// TIA Portal V18 program export: 2 tag tables, 0 data types, 2 data blocks, 3 code blocks (in call order from the OBs), 0 instance data blocks

VAR_GLOBAL   // PLC tag table "Default tag table"
   AD AT %MD6 : Real;
END_VAR

VAR_GLOBAL   // PLC tag table "PLC1_Tags"
   Start_Cmd AT %M0.0 : Bool;
   Stop_Cmd AT %M0.1 : Bool;
   bMotorRunning AT %M0.2 : Bool;
   Reset_Cmd AT %M0.3 : Bool;
   DIR_Cmd AT %M0.4 : Bool;
   PID_Setpoint AT %MD10 : Real;
   PID_ProcessValue AT %MD14 : Real;
   PID_Output AT %MD18 : Real;
   Speed_SP_toSend AT %MD22 : Real;
   Speed_PV_from2 AT %MD26 : Real;
   ATV12_Status AT %MW30 : Word;
   Control_Byte AT %MB32 : Byte;
   Clock_1Hz AT %M100.5 : Bool;
   GET_NDR AT %M1.0 : Bool;
   GET_Error AT %M1.1 : Bool;
   GET_Status AT %MW2 : Word;
   PUT_NDR AT %M1.2 : Bool;
   PUT_Error AT %M1.3 : Bool;
   PUT_Status AT %MW4 : Word;
END_VAR

DATA_BLOCK "DB10_NhanTuPLC2"   // DB10
{ S7_Optimized_Access := 'FALSE' }
VERSION : 0.1
// stored: AutoNumber true, IsOnlyStoredInLoadMemory false, IsWriteProtectedInAS false
   VAR
      Speed_Actual_fromPLC2 : Real;
      ATV12_Status_fromPLC2 : Word;
   END_VAR
BEGIN
END_DATA_BLOCK

DATA_BLOCK "DB11_GuiSangPLC2"   // DB11
{ S7_Optimized_Access := 'FALSE' }
VERSION : 0.1
// stored: AutoNumber true, IsOnlyStoredInLoadMemory false, IsWriteProtectedInAS false
   VAR
      Speed_SP_toSend : Real;
      Control_Byte_toSend : Bool;
      Reset_Cmd_toSend : Bool;
      DIR_Cmd_toSend : Bool;
   END_VAR
BEGIN
END_DATA_BLOCK

ORGANIZATION_BLOCK "Main"   // OB1, LAD, ProgramCycle
TITLE = "Main Program Sweep (Cycle)"
{ S7_Optimized_Access := 'TRUE' }
VERSION : 0.1
// stored: AutoNumber true, IsIECCheckEnabled false, SetENOAutomatically false
   VAR_INPUT
      Initial_Call : Bool;   // Initial call of this OB
      Remanence : Bool;   // =True, if remanent data are available
   END_VAR
BEGIN

REGION Network 1: Call FC_PLC1_Logic
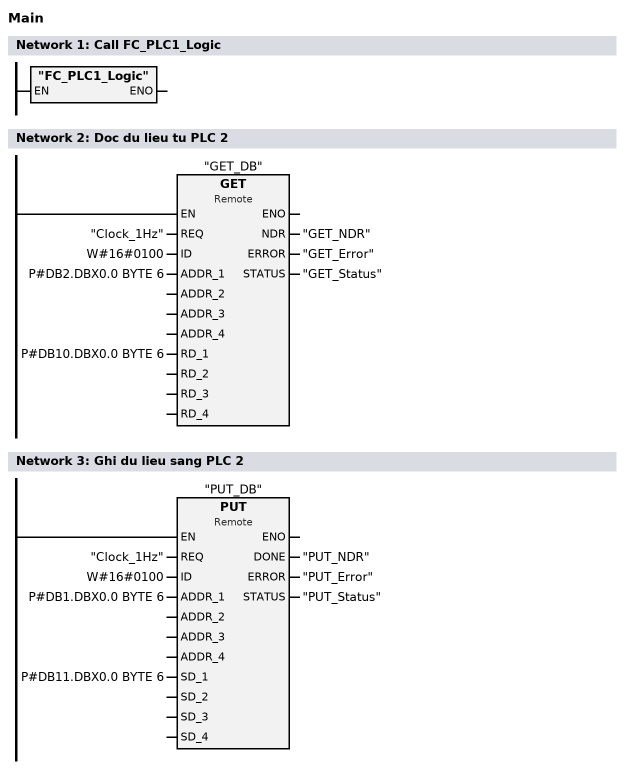
   RUNG wire#powerrail
      "FC_PLC1_Logic"()
   END_RUNG
   // the same network as SCL:
   "FC_PLC1_Logic"();
END_REGION

REGION Network 2: Doc du lieu tu PLC 2
   RUNG wire#powerrail
      { S7_Templates := "[remote_type := Remote, local_type := Variant]" } "GET_DB".GET(REQ := "Clock_1Hz", ID := W#16#0100, ADDR_1 := P#DB2.DBX0.0 BYTE 6, ADDR_2 :=, ADDR_3 :=, ADDR_4 :=, RD_1 := P#DB10.DBX0.0 BYTE 6, RD_2 :=, RD_3 :=, RD_4 :=, NDR => "GET_NDR", ERROR => "GET_Error", STATUS => "GET_Status")
   END_RUNG
   // the same network as SCL:
   "GET_DB"(REQ := "Clock_1Hz",   // GET
            ID := W#16#0100,
            ADDR_1 := P#DB2.DBX0.0 BYTE 6,
            RD_1 := P#DB10.DBX0.0 BYTE 6,
            NDR => "GET_NDR",
            ERROR => "GET_Error",
            STATUS => "GET_Status");
END_REGION

REGION Network 3: Ghi du lieu sang PLC 2
   RUNG wire#powerrail
      { S7_Templates := "[remote_type := Remote, local_type := Variant]" } "PUT_DB".PUT(REQ := "Clock_1Hz", ID := W#16#0100, ADDR_1 := P#DB1.DBX0.0 BYTE 6, ADDR_2 :=, ADDR_3 :=, ADDR_4 :=, SD_1 := P#DB11.DBX0.0 BYTE 6, SD_2 :=, SD_3 :=, SD_4 :=, DONE => "PUT_NDR", ERROR => "PUT_Error", STATUS => "PUT_Status")
   END_RUNG
   // the same network as SCL:
   "PUT_DB"(REQ := "Clock_1Hz",   // PUT
            ID := W#16#0100,
            ADDR_1 := P#DB1.DBX0.0 BYTE 6,
            SD_1 := P#DB11.DBX0.0 BYTE 6,
            DONE => "PUT_NDR",
            ERROR => "PUT_Error",
            STATUS => "PUT_Status");
END_REGION
END_ORGANIZATION_BLOCK

FUNCTION "FC_PLC1_Logic" : Void   // FC10, LAD
{ S7_Optimized_Access := 'TRUE' }
VERSION : 0.1
// stored: AutoNumber true, IsIECCheckEnabled false, SetENOAutomatically false, UDAEnableTagReadback false
BEGIN

REGION Network 1: Start Motor - Set bMotorRunning
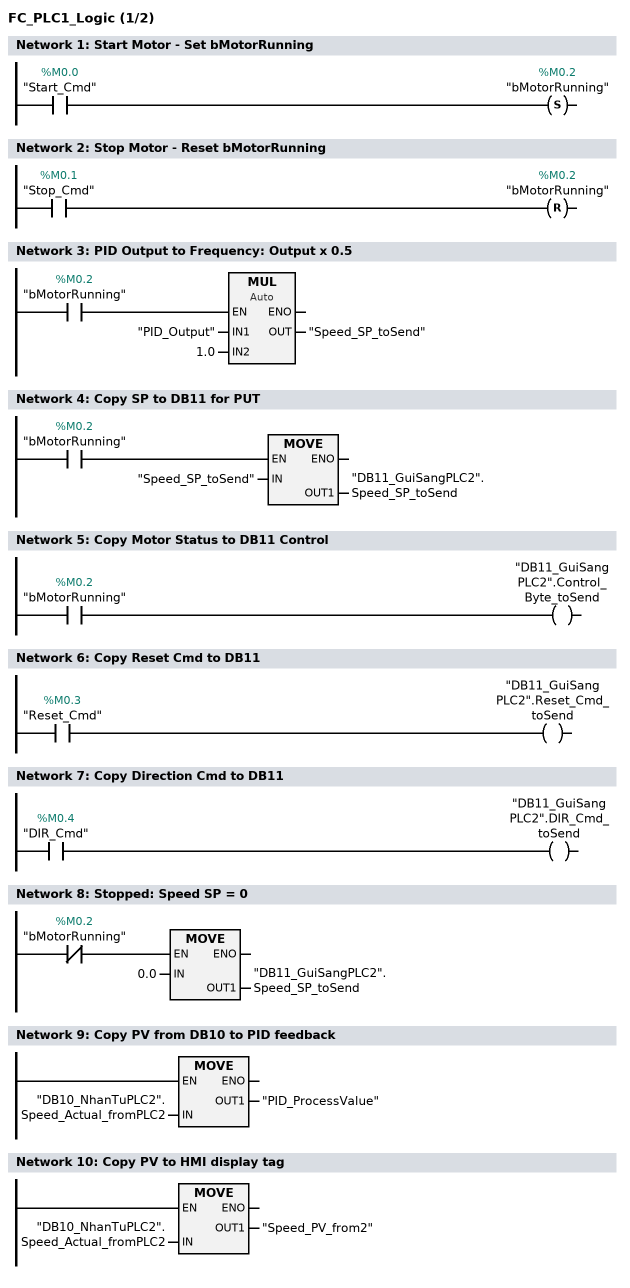
   RUNG wire#powerrail
      Contact( "Start_Cmd" )
      S_Coil( "bMotorRunning" )
   END_RUNG
   // the same network as SCL:
   IF "Start_Cmd" THEN "bMotorRunning" := TRUE; END_IF;
END_REGION

REGION Network 2: Stop Motor - Reset bMotorRunning
   RUNG wire#powerrail
      Contact( "Stop_Cmd" )
      R_Coil( "bMotorRunning" )
   END_RUNG
   // the same network as SCL:
   IF "Stop_Cmd" THEN "bMotorRunning" := FALSE; END_IF;
END_REGION

REGION Network 3: PID Output to Frequency: Output x 0.5
   RUNG wire#powerrail
      Contact( "bMotorRunning" )
      { S7_GenerateENO := "TRUE" } Mul(in1 := "PID_Output", in2 := 1.0, out => "Speed_SP_toSend")
   END_RUNG
   // the same network as SCL:
   IF "bMotorRunning" THEN "Speed_SP_toSend" := "PID_Output" * 1.0; END_IF;
END_REGION

REGION Network 4: Copy SP to DB11 for PUT
   RUNG wire#powerrail
      Contact( "bMotorRunning" )
      { S7_GenerateENO := "TRUE" } Move(in := "Speed_SP_toSend", out1 => "DB11_GuiSangPLC2".Speed_SP_toSend)
   END_RUNG
   // the same network as SCL:
   IF "bMotorRunning" THEN "DB11_GuiSangPLC2".Speed_SP_toSend := "Speed_SP_toSend"; END_IF;
END_REGION

REGION Network 5: Copy Motor Status to DB11 Control
   RUNG wire#powerrail
      Contact( "bMotorRunning" )
      Coil( "DB11_GuiSangPLC2".Control_Byte_toSend )
   END_RUNG
   // the same network as SCL:
   "DB11_GuiSangPLC2".Control_Byte_toSend := "bMotorRunning";
END_REGION

REGION Network 6: Copy Reset Cmd to DB11
   RUNG wire#powerrail
      Contact( "Reset_Cmd" )
      Coil( "DB11_GuiSangPLC2".Reset_Cmd_toSend )
   END_RUNG
   // the same network as SCL:
   "DB11_GuiSangPLC2".Reset_Cmd_toSend := "Reset_Cmd";
END_REGION

REGION Network 7: Copy Direction Cmd to DB11
   RUNG wire#powerrail
      Contact( "DIR_Cmd" )
      Coil( "DB11_GuiSangPLC2".DIR_Cmd_toSend )
   END_RUNG
   // the same network as SCL:
   "DB11_GuiSangPLC2".DIR_Cmd_toSend := "DIR_Cmd";
END_REGION

REGION Network 8: Stopped: Speed SP = 0
   RUNG wire#powerrail
      I_Contact( "bMotorRunning" )
      { S7_GenerateENO := "TRUE" } Move(in := 0.0, out1 => "DB11_GuiSangPLC2".Speed_SP_toSend)
   END_RUNG
   // the same network as SCL:
   IF NOT "bMotorRunning" THEN "DB11_GuiSangPLC2".Speed_SP_toSend := 0.0; END_IF;
END_REGION

REGION Network 9: Copy PV from DB10 to PID feedback
   RUNG wire#powerrail
      { S7_GenerateENO := "TRUE" } Move(in := "DB10_NhanTuPLC2".Speed_Actual_fromPLC2, out1 => "PID_ProcessValue")
   END_RUNG
   // the same network as SCL:
   "PID_ProcessValue" := "DB10_NhanTuPLC2".Speed_Actual_fromPLC2;
END_REGION

REGION Network 10: Copy PV to HMI display tag
   RUNG wire#powerrail
      { S7_GenerateENO := "TRUE" } Move(in := "DB10_NhanTuPLC2".Speed_Actual_fromPLC2, out1 => "Speed_PV_from2")
   END_RUNG
   // the same network as SCL:
   "Speed_PV_from2" := "DB10_NhanTuPLC2".Speed_Actual_fromPLC2;
END_REGION

REGION Network 11: Copy ATV12 Status to HMI tag
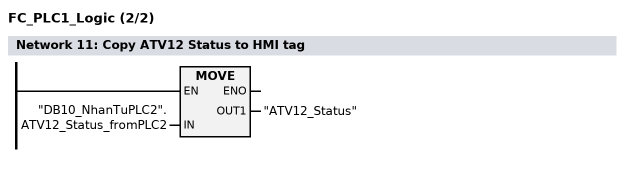
   RUNG wire#powerrail
      { S7_GenerateENO := "TRUE" } Move(in := "DB10_NhanTuPLC2".ATV12_Status_fromPLC2, out1 => "ATV12_Status")
   END_RUNG
   // the same network as SCL:
   "ATV12_Status" := "DB10_NhanTuPLC2".ATV12_Status_fromPLC2;
END_REGION
END_FUNCTION

ORGANIZATION_BLOCK "Cyclic interrupt"   // OB30, LAD, CyclicInterrupt
{ S7_Optimized_Access := 'TRUE' }
VERSION : 0.1
// stored: AutoNumber true, IsIECCheckEnabled false, SetENOAutomatically false
   VAR_INPUT
      Initial_Call : Bool;   // Initial call of this OB
      Event_Count : Int;   // Events discarded
   END_VAR
BEGIN

REGION Network 1
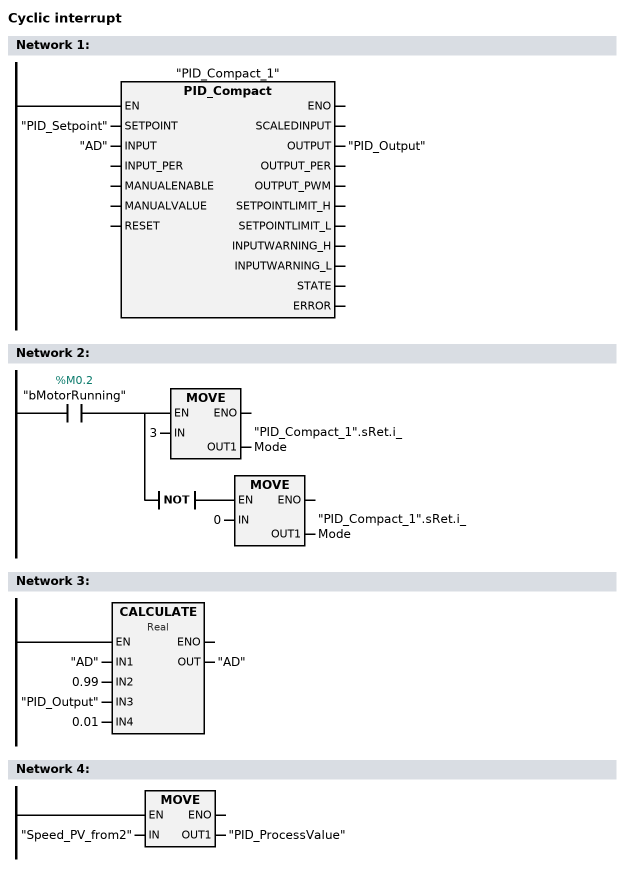
   RUNG wire#powerrail
      "PID_Compact_1".PID_Compact(Setpoint := "PID_Setpoint", Input := "AD", Input_PER :=, ManualEnable :=, ManualValue :=, Reset :=, ScaledInput =>, Output => "PID_Output", Output_PER =>, Output_PWM =>, SetpointLimit_H =>, SetpointLimit_L =>, InputWarning_H =>, InputWarning_L =>, State =>, Error =>)
   END_RUNG
   // the same network as SCL:
   "PID_Compact_1"(Setpoint := "PID_Setpoint", Input := "AD", Output => "PID_Output");   // PID_Compact
END_REGION

REGION Network 2
   RUNG wire#powerrail
      Contact( "bMotorRunning" )
      wire#w1
      Move(in := 3, out1 => "PID_Compact_1".sRet.i_Mode)
   END_RUNG
   RUNG wire#w1
      Not()
      Move(in := 0, out1 => "PID_Compact_1".sRet.i_Mode)
   END_RUNG
   // the same network as SCL:
   IF "bMotorRunning" THEN "PID_Compact_1".sRet.i_Mode := 3; END_IF;
   IF NOT "bMotorRunning" THEN "PID_Compact_1".sRet.i_Mode := 0; END_IF;
END_REGION

REGION Network 3
   RUNG wire#powerrail
      { S7_Templates := "SrcType := Real"; S7_Expression := "IN2*IN1 + IN4*IN3" } Calculate(in1 := "AD", in2 := 0.99, in3 := "PID_Output", in4 := 0.01, out => "AD")
   END_RUNG
   // the same network as SCL:
   "AD" := 0.99*"AD" + 0.01*"PID_Output";
END_REGION

REGION Network 4
   RUNG wire#powerrail
      Move(in := "Speed_PV_from2", out1 => "PID_ProcessValue")
   END_RUNG
   // the same network as SCL:
   "PID_ProcessValue" := "Speed_PV_from2";
END_REGION
END_ORGANIZATION_BLOCK
